FUNCTION_BLOCK FB_RAT
VAR_INPUT
END_VAR
VAR_OUTPUT
END_VAR
VAR
END_VAR

END_FUNCTION_BLOCK

(* stored: Version 1.1.0.1, ProductVersion 3.1.4024.16
   POU FB_RAT: Id {a53e8369-ccc0-4a67-aaae-0302ede3efed}, SpecialFunc None *)
